% RSLogix 500 project LAB3.RSS, saved by version 8.10.00.30 %
PROJECT "LAB3"    % processor: Bul.1763 MicroLogix 1100 Series A %

PROGRAM FILES
  LAD 2   9 rungs

DATA FILES
  O0 OUTPUT  4 elements
  I1 INPUT  6 elements
  S2 STATUS  66 elements
  B3 BINARY  1 elements
  T4 TIMER  1 elements
  C5 COUNTER  1 elements
  R6 CONTROL  1 elements
  N7 INTEGER  1 elements
  F8 FLOAT  1 elements

LADDER 2
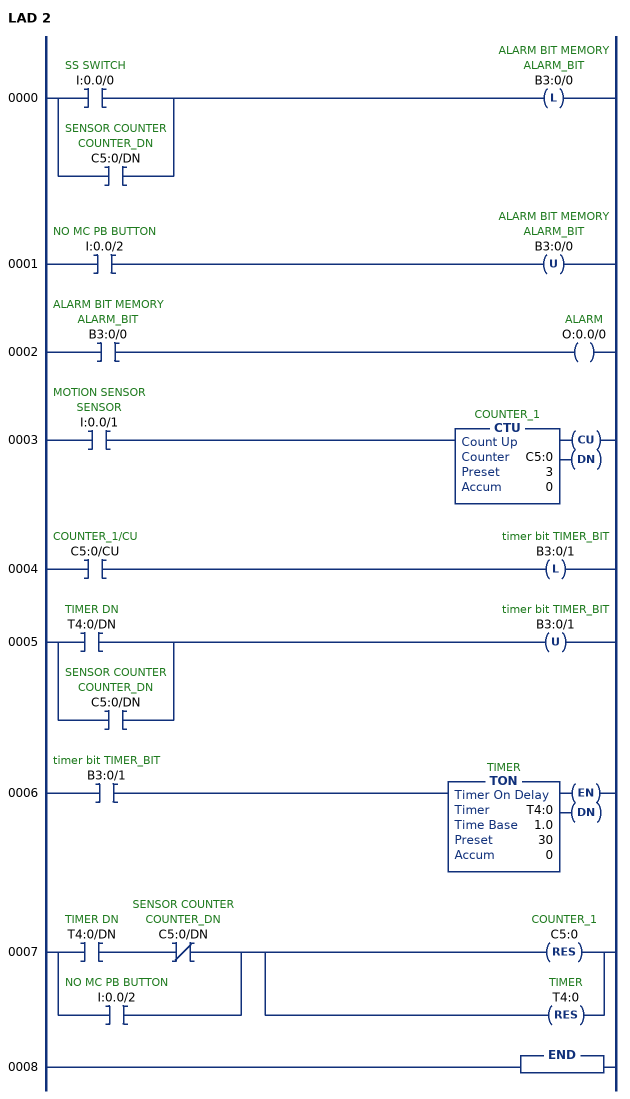
% Rung: 0 %
SOR BST XIC I:0.0/0 NXB XIC C5:0/DN BND OTL B3:0/0 EOR
%   I:0.0/0  SWITCH  "SS" %
%   C5:0/DN  COUNTER_DN  "SENSOR COUNTER" %
%   B3:0/0  ALARM_BIT  "ALARM BIT MEMORY" %
% Rung: 1 %
SOR XIC I:0.0/2 OTU B3:0/0 EOR
%   I:0.0/2  BUTTON  "NO MC PB" %
%   B3:0/0  ALARM_BIT  "ALARM BIT MEMORY" %
% Rung: 2 %
SOR XIC B3:0/0 OTE O:0.0/0 EOR
%   B3:0/0  ALARM_BIT  "ALARM BIT MEMORY" %
%   O:0.0/0  ALARM %
% Rung: 3 %
SOR XIC I:0.0/1 CTU C5:0 3 0 EOR
%   I:0.0/1  SENSOR  "MOTION SENSOR" %
%   C5:0  COUNTER_1 %
% Rung: 4 %
SOR XIC C5:0/CU OTL B3:0/1 EOR
%   C5:0  COUNTER_1 %
%   B3:0/1  TIMER_BIT  "timer bit" %
% Rung: 5 %
SOR BST XIC T4:0/DN NXB XIC C5:0/DN BND OTU B3:0/1 EOR
%   T4:0/DN  "TIMER DN" %
%   C5:0/DN  COUNTER_DN  "SENSOR COUNTER" %
%   B3:0/1  TIMER_BIT  "timer bit" %
% Rung: 6 %
SOR XIC B3:0/1 TON T4:0 1.0 30 0 EOR
%   B3:0/1  TIMER_BIT  "timer bit" %
%   T4:0  "TIMER" %
% Rung: 7 %
SOR BST XIC T4:0/DN XIO C5:0/DN NXB XIC I:0.0/2 BND BST RES C5:0 NXB RES T4:0 BND EOR
%   T4:0/DN  "TIMER DN" %
%   C5:0/DN  COUNTER_DN  "SENSOR COUNTER" %
%   I:0.0/2  BUTTON  "NO MC PB" %
%   C5:0  COUNTER_1 %
%   T4:0  "TIMER" %
% Rung: 8 %
SOR END EOR

OTHER DOCUMENTED ADDRESSES
  C5:0/0  COUNTER  "MOTION SENSOR (3)"
  I:0.0/3  "MOTION SENSOR"
  I:0.0/6  L_2
  T4:0/EN  TIMER

DATA TABLE (non-zero values as saved)
DATA T4
% .PRE .ACC %
% T4:0 % 30 0
DATA C5
% .PRE .ACC %
% C5:0 % 3 0
